(* LS Electric XG5000 project: 241008_연습문제 *)
(* PLC LSPLC *)
(* module base 0 slot 0: 입력 모듈:XGI-D21A (DC 24V 입력, 8점 (전류소스/싱크입력)) *)
(* module base 0 slot 1: 출력 모듈:XGQ-RY1A (릴레이 출력, 8점 (2A용, 단독 COM.)) *)

PROGRAM NewProgram (* task: 스캔 프로그램 *)
VAR
    P1 AT %IX0.0.0 : BOOL;
    P10 AT %QX0.1.1 : BOOL;
    P11 AT %QX0.1.0 : BOOL;
END_VAR

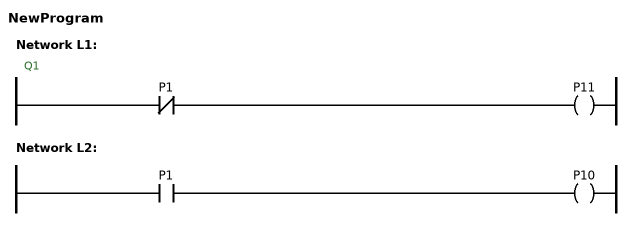
(* Q1 *)
(* Rung L1 *)
P11 := NOT P1;
(* Rung L2 *)
P10 := P1;
END_PROGRAM